(**************************************************************************************
 * 	Application		:	BoxControl Framework
 *	Revision		:	$Revision: 404529 $
 *	Revision date	:	$Date: 2018-04-23 08:21:38 +0200 (Mo., 23 Apr 2018) $
 *	Last changed by	:	$Author: b7bolm $
 *	URL				:	$URL: http://almscdc.swisslog.com/repo/SWPD/Development/BoxControlFramework/20_Release/trunk/01_Software/BCF/BCF/JumpStart/20_Product/11_Emu/10_Base/10_Lib/00_GVLs/SystemEmulation.TcGVL $
 *
 *	Purpose			:	Base emulation global variables.
 *
 * ------------------------------------------------------------------------------------
 *	Copyright Swisslog [IP AG], Switzerland. All rights reserved.
 * 
 * ------------------------------------------------------------------------------------
 *	
 * 	Revision History: 
 *
 * 	VERSION			DATE			INITIALS			DESCRIPTION
 *	0.1				01.01.2001		swl					Example
 *
 **************************************************************************************)
VAR_GLOBAL
	fbMFCS_ChannelEmulation		: ARRAY [E_MFCS_Channel.BEGIN_CHANNEL .. E_MFCS_Channel.END_CHANNEL] OF ITF_MFCS_Emulation; // MFCS connections
	fbITC_ManagerEmulation		: ITF_ITC_Emulation;
END_VAR

(* stored: Version 1.1.0.1, ProductVersion 3.1.4022.12
   GVL SystemEmulation: Id {9aedf1ed-7dbe-4fc8-bc86-44972e176549} *)
